FUNCTION_BLOCK SledgeHAL (* Composite Function Block Type *)
  (* Standard: 61499-2 *)
  (* Version 0.0, 9/26/2018, dmidro, nxtControl GmbH, template *)
  PACKAGE Main;
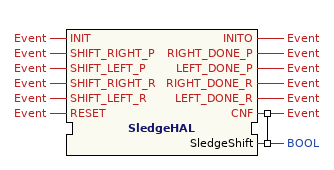
  EVENT_INPUT
    INIT; (* Initialization Request *)
    SHIFT_RIGHT_P; (* Set Event *)
    SHIFT_LEFT_P; (* Reset Event *)
    SHIFT_RIGHT_R;
    SHIFT_LEFT_R;
    RESET; (* Reset Event *)
  END_EVENT
  EVENT_OUTPUT
    INITO; (* Initialization Confirm *)
    RIGHT_DONE_P; (* Delayed Event *)
    LEFT_DONE_P; (* Delayed Event *)
    RIGHT_DONE_R;
    LEFT_DONE_R;
    CNF WITH SledgeShift;
  END_EVENT
  VAR_OUTPUT
    SledgeShift : BOOL; (* Current Output State *)
  END_VAR
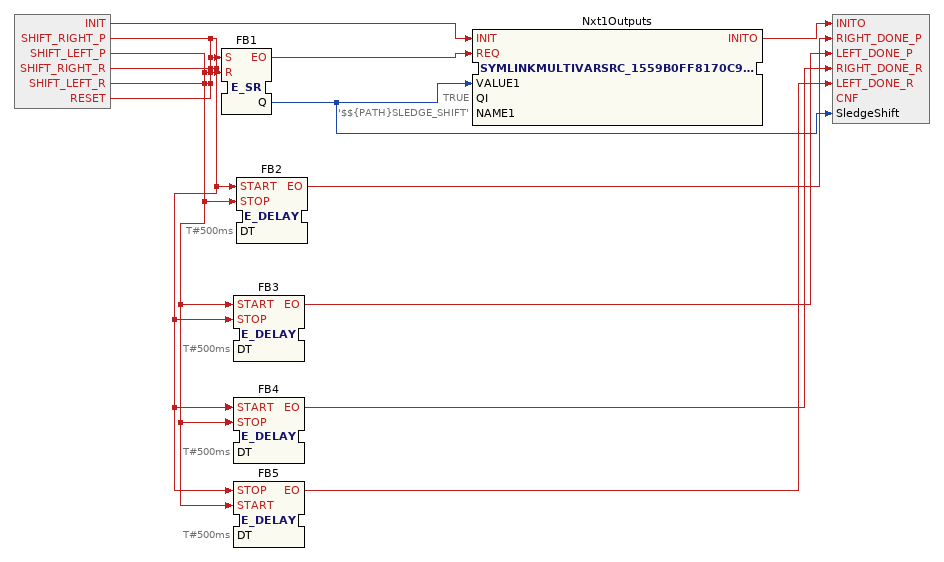
  FBS
    Nxt1Outputs : SYMLINKMULTIVARSRC_1559B0FF8170C9BA0(QI := TRUE, NAME1 := '$${PATH}SLEDGE_SHIFT'); {SET_ATTRIBUTE(Configuration.GenericFBType.InterfaceParams, Runtime.System#I:=1;VALUE${I$}:BOOL)}
    FB1 : E_SR;
    FB2 : E_DELAY(DT := T#500ms);
    FB3 : E_DELAY(DT := T#500ms);
    FB4 : E_DELAY(DT := T#500ms);
    FB5 : E_DELAY(DT := T#500ms);
  END_FBS
  EVENT_CONNECTIONS
    INIT TO Nxt1Outputs.INIT;
    Nxt1Outputs.INITO TO INITO;
    SHIFT_RIGHT_P TO FB1.S;
    SHIFT_LEFT_P TO FB1.R;
    FB1.EO TO Nxt1Outputs.REQ;
    FB2.EO TO RIGHT_DONE_P;
    FB3.EO TO LEFT_DONE_P;
    SHIFT_RIGHT_P TO FB2.START;
    SHIFT_LEFT_P TO FB2.STOP;
    SHIFT_LEFT_P TO FB3.START;
    SHIFT_RIGHT_P TO FB3.STOP;
    RESET TO FB1.R;
    FB4.EO TO RIGHT_DONE_R;
    FB5.EO TO LEFT_DONE_R;
    SHIFT_RIGHT_R TO FB4.START;
    SHIFT_RIGHT_R TO FB5.STOP;
    SHIFT_LEFT_R TO FB4.STOP;
    SHIFT_LEFT_R TO FB5.START;
    SHIFT_RIGHT_R TO FB1.S;
    SHIFT_LEFT_R TO FB1.R;
  END_CONNECTIONS
  DATA_CONNECTIONS
    FB1.Q TO Nxt1Outputs.VALUE1;
    FB1.Q TO SledgeShift;
  END_CONNECTIONS
END_FUNCTION_BLOCK
